// TIA Portal project "ObjectArray" (V16)

(* hardware
DEVICE "ET 200SP station_1"  ET 200SP-Station
   slot 0: "Rack_0"  Rack  6ES5 710-8MAx1
   slot 1: "PLC_1"  CPU 1510SP-1 PN  6ES7 510-1DJ00-0AB0  V1.8
      slot 32768: "PROFINET interface_1"  X1
         slot 32771: "Port_3"  X1 P3
   slot 2: "Server module_1"  Server module  6ES7 193-6PA00-0AA0  V1.1
      slot 1: "Server module_1"  Server module
   slot 127: "BA 2xRJ45"  BA 2xRJ45  6ES7 193-6AR00-0AA0  V0.0
      slot 32769: "Port_1"  X1 P1  6ES7 193-6AR00-0AA0
      slot 32770: "Port_2"  X1 P2  6ES7 193-6AR00-0AA0
*)

// ===== PLC "PLC_1"  CPU 1510SP-1 PN =====

// folder: ContactorDataType

TYPE "tyContactor_Input"
   STRUCT
      bContactorStartRequest : Bool;
      bContactorFeedbackInput : Bool;
   END_STRUCT;
END_TYPE

TYPE "tyContactor_Output"
   STRUCT
      bActivateContactorCoil : Bool;
      bContactorFault : Bool;
      b_MotorIsRunning : Bool;
   END_STRUCT;
END_TYPE

TYPE "tyContactor_StaticData"
   STRUCT
      TContactorControllTimer : TON_TIME;
      TcontactorFeedBackControlTime : Time;
   END_STRUCT;
END_TYPE

TYPE "tyContactor_Main"
   STRUCT
      ContactorInputs : "tyContactor_Input";
      ContactorOutputs : "tyContactor_Output";
      ContactorStatic : "tyContactor_StaticData";
   END_STRUCT;
END_TYPE

// folder: (top level)

DATA_BLOCK "ContactorControll_Obj_DB"   // DB1
{ S7_Optimized_Access := 'TRUE' }
VERSION : 0.1
// stored: InstanceOfName ContactorControll_Obj
"ContactorControll_Obj"
BEGIN
END_DATA_BLOCK

FUNCTION_BLOCK "ContactorControll_Obj"   // FB1, SCL
{ S7_Optimized_Access := 'TRUE' }
VERSION : 0.1
   VAR
      MotorContactorControll : Array[0..10] of "tyContactor_Main";
   END_VAR
   VAR_TEMP
      i : Int;
   END_VAR
BEGIN
   //=============================================================================
   // Dmitri Raihtsaum - Copyright 2023
   // Created By: Dmitri Raihtsaum
   //-----------------------------------------------------------------------------
   // Tested with:   CPU 1510SP-1 PN
   // Engineering:   TIA Portal V16
   // Functionality: Contactor Control Object 
   // Date: 09.04.2023
   // Rev 0.1
   //=============================================================================

   FOR #i := 0 TO 10 DO

       //Mapping
       #MotorContactorControll[#i].ContactorStatic.TcontactorFeedBackControlTime := t#2s;
       //Logic
       //Contactor Start signal 
       IF #MotorContactorControll[#i].ContactorInputs.bContactorStartRequest THEN
           #MotorContactorControll[#i].ContactorOutputs.bActivateContactorCoil := TRUE;
       END_IF;
       //Contactor Stop signal
       IF NOT #MotorContactorControll[#i].ContactorInputs.bContactorStartRequest THEN
           #MotorContactorControll[#i].ContactorOutputs.bActivateContactorCoil := FALSE;
       END_IF;
       //Check Contactor Status 
       IF #MotorContactorControll[#i].ContactorOutputs.bActivateContactorCoil AND #MotorContactorControll[#i].ContactorInputs.bContactorFeedbackInput THEN
           #MotorContactorControll[#i].ContactorOutputs.b_MotorIsRunning := TRUE;
       ELSE
           #MotorContactorControll[#i].ContactorOutputs.b_MotorIsRunning := FALSE;
       END_IF;
       // Fault Signal
       IF #MotorContactorControll[#i].ContactorInputs.bContactorStartRequest AND NOT #MotorContactorControll[#i].ContactorInputs.bContactorFeedbackInput
           OR NOT #MotorContactorControll[#i].ContactorInputs.bContactorStartRequest AND #MotorContactorControll[#i].ContactorInputs.bContactorFeedbackInput
       THEN
           #MotorContactorControll[#i].ContactorStatic.TContactorControllTimer(IN := TRUE,
                                                                               PT := #MotorContactorControll[#i].ContactorStatic.TcontactorFeedBackControlTime);
       ELSE
           #MotorContactorControll[#i].ContactorStatic.TContactorControllTimer(IN := FALSE,
                                                                               PT := t#0ms);
       END_IF;
       // Fault Flag
       IF #MotorContactorControll[#i].ContactorStatic.TContactorControllTimer.Q THEN
           #MotorContactorControll[#i].ContactorOutputs.bContactorFault := TRUE;
       ELSE
           #MotorContactorControll[#i].ContactorOutputs.bContactorFault := FALSE;
       END_IF;
   END_FOR;
   //=============================================================================
   //END
   //=============================================================================
END_FUNCTION_BLOCK

ORGANIZATION_BLOCK "Main"   // OB1, LAD, ProgramCycle
TITLE = "Main Program Sweep (Cycle)"
{ S7_Optimized_Access := 'TRUE' }
VERSION : 0.1
   VAR_INPUT
      Initial_Call : Bool;   // Initial call of this OB
      Remanence : Bool;   // =True, if remanent data are available
   END_VAR
BEGIN

REGION Network 1
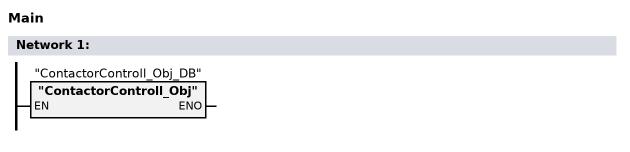
   RUNG wire#powerrail
      "ContactorControll_Obj_DB"()
   END_RUNG
   // the same network as SCL:
   "ContactorControll_Obj_DB"();   // "ContactorControll_Obj"
END_REGION
END_ORGANIZATION_BLOCK